{attribute 'qualified_only'}
VAR_GLOBAL
	// Pitch Mechanism:
	{attribute 'TcLinkTo' := '.diEncCnt:=TIIB[EL5042_XRTM1_PitchBender]^FB Inputs Channel 1^Position'}
	XRTM1_Pitch : HOMS_PitchMechanism := (ReqPosLimHi := 120.0,
		                                 ReqPosLimLo := -182.0,
		                                 diEncPosLimHi := 8662020,
		                                 diEncPosLimLo := 8507095);
END_VAR

(* stored: Version 1.1.0.1, ProductVersion 3.1.4022.18
   GVL GVL_XRTM1: Id {c3e91af1-5ac0-497f-aea6-a43e8c284355} *)
